% RSLogix 500 project MAGAZYN.rss, saved by version 8.30.00.16 %
PROJECT "SPRAWKO1"    % processor: Bul.1763 MicroLogix 1100 Series B %

PROGRAM FILES
  LAD 2   13 rungs

DATA FILES
  O0 OUTPUT  4 elements
  I1 INPUT  6 elements
  S2 STATUS  66 elements
  B3 BINARY  10 elements
  T4 TIMER  10 elements
  C5 COUNTER  1 elements
  R6 CONTROL  1 elements
  N7 INTEGER  10 elements
  F8 FLOAT  1 elements

LADDER 2
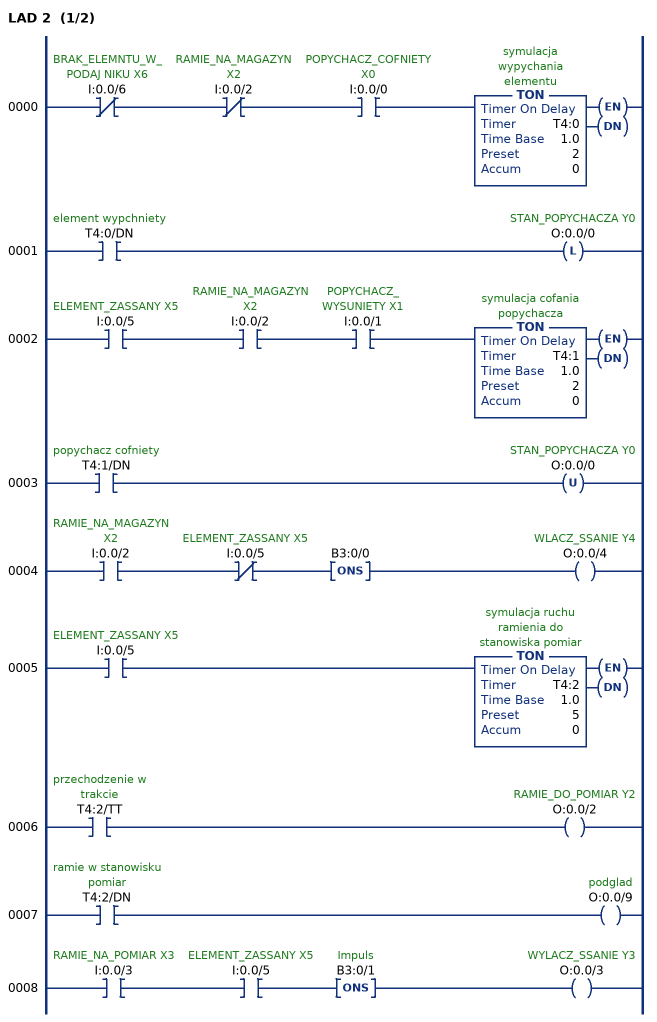
% Rung: 0 %
SOR XIO I:0.0/6 XIO I:0.0/2 XIC I:0.0/0 TON T4:0 1.0 2 0 EOR
%   I:0.0/6  X6  "BRAK_ELEMNTU_W_PODAJ NIKU" %
%   I:0.0/2  X2  "RAMIE_NA_MAGAZYN" %
%   I:0.0/0  X0  "POPYCHACZ_COFNIETY" %
%   T4:0  "symulacja wypychania elementu" %
% Rung: 1 %
SOR XIC T4:0/DN OTL O:0.0/0 EOR
%   T4:0/DN  "element wypchniety" %
%   O:0.0/0  Y0  "STAN_POPYCHACZA" %
% Rung: 2 %
SOR XIC I:0.0/5 XIC I:0.0/2 XIC I:0.0/1 TON T4:1 1.0 2 0 EOR
%   I:0.0/5  X5  "ELEMENT_ZASSANY" %
%   I:0.0/2  X2  "RAMIE_NA_MAGAZYN" %
%   I:0.0/1  X1  "POPYCHACZ_WYSUNIETY" %
%   T4:1  "symulacja cofania popychacza" %
% Rung: 3 %
SOR XIC T4:1/DN OTU O:0.0/0 EOR
%   T4:1/DN  "popychacz cofniety" %
%   O:0.0/0  Y0  "STAN_POPYCHACZA" %
% Rung: 4 %
SOR XIC I:0.0/2 XIO I:0.0/5 ONS B3:0/0 OTE O:0.0/4 EOR
%   I:0.0/2  X2  "RAMIE_NA_MAGAZYN" %
%   I:0.0/5  X5  "ELEMENT_ZASSANY" %
%   O:0.0/4  Y4  "WLACZ_SSANIE" %
% Rung: 5 %
SOR XIC I:0.0/5 TON T4:2 1.0 5 0 EOR
%   I:0.0/5  X5  "ELEMENT_ZASSANY" %
%   T4:2  "symulacja ruchu ramienia do stanowiska pomiar" %
% Rung: 6 %
SOR XIC T4:2/TT OTE O:0.0/2 EOR
%   T4:2/TT  "przechodzenie w trakcie" %
%   O:0.0/2  Y2  "RAMIE_DO_POMIAR" %
% Rung: 7 %
SOR XIC T4:2/DN OTE O:0.0/9 EOR
%   T4:2/DN  "ramie w stanowisku pomiar" %
%   O:0.0/9  "podglad" %
% Rung: 8 %
SOR XIC I:0.0/3 XIC I:0.0/5 ONS B3:0/1 OTE O:0.0/3 EOR
%   I:0.0/3  X3  "RAMIE_NA_POMIAR" %
%   I:0.0/5  X5  "ELEMENT_ZASSANY" %
%   B3:0/1  "Impuls" %
%   O:0.0/3  Y3  "WYLACZ_SSANIE" %

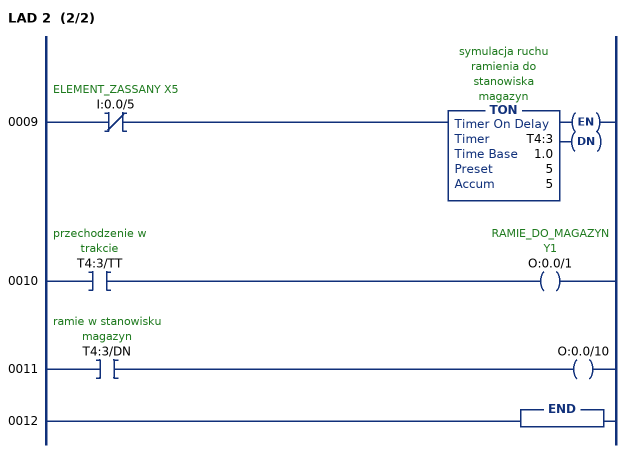
% Rung: 9 %
SOR XIO I:0.0/5 TON T4:3 1.0 5 5 EOR
%   I:0.0/5  X5  "ELEMENT_ZASSANY" %
%   T4:3  "symulacja ruchu ramienia do stanowiska magazyn" %
% Rung: 10 %
SOR XIC T4:3/TT OTE O:0.0/1 EOR
%   T4:3/TT  "przechodzenie w trakcie" %
%   O:0.0/1  Y1  "RAMIE_DO_MAGAZYN" %
% Rung: 11 %
SOR XIC T4:3/DN OTE O:0.0/10 EOR
%   T4:3/DN  "ramie w stanowisku magazyn" %
% Rung: 12 %
SOR END EOR

OTHER DOCUMENTED ADDRESSES
  T4:0/0  "Wysuwanie popychacza"
  T4:0/1  "Cofniecie popychacza"

DATA TABLE (non-zero values as saved)
DATA B3
% B3:0 % 0X0005 0X0000 0X0000 0X0000 0X0000 0X0000 0X0000 0X0000 0X0000 0X0000
DATA T4
% .PRE .ACC %
% T4:0 % 2 0
% T4:1 % 2 0
% T4:2 % 5 0
% T4:3 % 5 5
